// Mitsubishi GX Works2 project: plc_group6   PLC: FX3G

// global labels: Global1
VAR_GLOBAL
  switch10 AT X010 : BOOL;
  machineA AT M0 : BOOL;
  close_sys AT X005 : BOOL;
  sen_1 AT X001 : BOOL;
  sen_30 AT X002 : BOOL;
  sen_15 AT X003 : BOOL;
  sen_2 AT X004 : BOOL;
  zeluf_on AT Y004 : BOOL;
END_VAR
VAR_GLOBAL CONSTANT
  cream : INT := 700;
  chocolate : INT := 500;
  biscuit : INT := 100;
  ZeroConst : REAL;
END_VAR
VAR_GLOBAL
  TS1 : BOOL;
  TC1 AT TC1 : BOOL;
END_VAR
VAR_GLOBAL CONSTANT
  sec : INT := 40;
  sec_4 : INT := 40;
END_VAR
VAR_GLOBAL
  coil_y0 AT Y000 : BOOL;
  blink1 AT TS1 : BOOL;
  blink AT TC1 : BOOL;
  blink2 AT TC2 : BOOL;
  blink3 AT TS2 : BOOL;
  coil_y1 AT Y001 : BOOL;
  D_cream AT D1100 : REAL;
  D_chocolate AT D1102 : REAL;
  D_biscuit AT D1104 : REAL;
  end_day AT M1 : BOOL;
  start_day_button AT X007 : BOOL;
  start AT M2 : BOOL;
  start_day_lamp AT Y007 : BOOL;
  timer_tc3 AT TC3 : BOOL;
END_VAR
VAR_GLOBAL CONSTANT
  const_30_sec : INT := 30;
END_VAR
VAR_GLOBAL
  timer_ts3 AT TS3 : BOOL;
  blink_end AT M3 : BOOL;
END_VAR
VAR_GLOBAL CONSTANT
  cream_300 : REAL := 300;
  chocolate_240 : REAL := 240;
  biscuit_6 : REAL := 6;
END_VAR
VAR_GLOBAL
  D_ziluf AT D1106 : REAL;
  ziluf_button_x11 AT X011 : BOOL;
  ziluf_finish AT M4 : BOOL;
  D_tvila AT D1108 : REAL;
  sample_batton_x6 AT X006 : BOOL;
END_VAR
VAR_GLOBAL CONSTANT
  cream_700 : REAL := 700;
  chocolate_500 : REAL := 500;
  biscuit_100 : REAL := 100;
  nomalization : REAL := 400;
  nomalization_400 : REAL := 400;
END_VAR
VAR_GLOBAL
  sample_finish AT M5 : BOOL;
  finish_tvila_lamp AT Y003 : BOOL;
END_VAR
VAR_GLOBAL CONSTANT
  Double_tvila : REAL := 5;
  Double_amount : REAL := 240;
  normal_amount : REAL := 120;
END_VAR
VAR_GLOBAL
  timer_tc4 AT TC4 : BOOL;
END_VAR
VAR_GLOBAL CONSTANT
  sec_5 : INT := 50;
END_VAR
VAR_GLOBAL
  time_ts4 AT TS4 : BOOL;
  analog_input_1 AT D8280 : INT;
  blink_m5 AT M5 : BOOL;
  blink_m6 AT M6 : BOOL;
  data_analog_input_1 AT D1112 : INT;
  finish_tvila AT M7 : BOOL;
  start_ariza AT X000 : BOOL;
  counter_ariza_krembo AT CC0 : BOOL;
END_VAR
VAR_GLOBAL CONSTANT
  krembo_ariza_5 : INT := 5;
END_VAR
VAR_GLOBAL
  counter_ariza_krembo_5 AT CS0 : BOOL;
  counter_ariza_krembo_5_lamp AT Y002 : BOOL;
  counter_ariza_stop AT M8 : BOOL;
  krembo_sum AT D1114 : REAL;
END_VAR
VAR_GLOBAL CONSTANT
  add_krembo : REAL := 1;
END_VAR
VAR_GLOBAL
  counter_ariza_krembo_6 AT CC1 : BOOL;
END_VAR
VAR_GLOBAL CONSTANT
  krembo_ariza_6 : INT := 6;
END_VAR
VAR_GLOBAL
  check_stock AT M12 : BOOL;
END_VAR
VAR_GLOBAL CONSTANT
  multiply : INT := 40;
END_VAR
VAR_GLOBAL
  analog_output AT D8282 : INT;
  cream_input AT D1116 : REAL;
  chocolate_input AT D1118 : REAL;
  biscuit_input AT D1120 : REAL;
END_VAR
VAR_GLOBAL CONSTANT
  blink5 : INT := 5;
END_VAR
VAR_GLOBAL
  timer_tc5 AT TC5 : BOOL;
  help_blink1 AT M9 : BOOL;
  help_blink2 AT M10 : BOOL;
  help_blink3 AT M11 : BOOL;
  blink_tc6 AT TC6 : BOOL;
  blink_ts6 AT TS6 : BOOL;
  blink_tc7 AT TC7 : BOOL;
  blink_ts7 AT TS7 : BOOL;
  counter_ariza_krembo_6_stop AT CS1 : BOOL;
  sample AT D1121 : REAL;
END_VAR

// task Task_01 (event TRUE, interval 0, priority 31): POU_01

PROGRAM POU_01
VAR CONSTANT
  timer_ts4 : BOOL;
END_VAR
(* structured ladder/FBD written out as ST: instructions are called as NAME(EN, inputs, outputs); _pN, _eN, _tN stand for wires *)
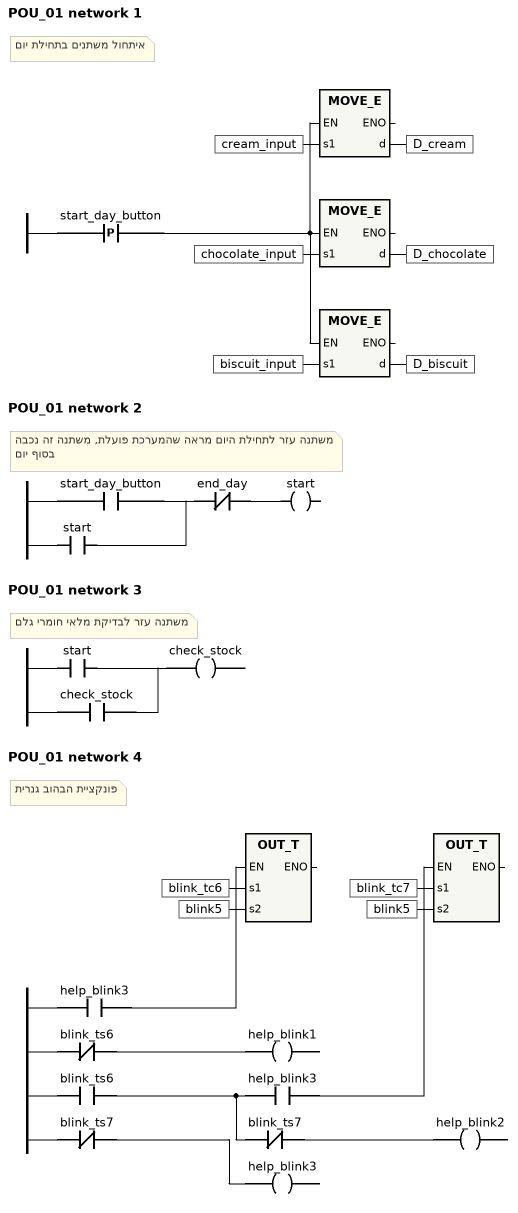
(* network 1 *)
(* איתחול משתנים בתחילת יום *)
_p1 := LDP(TRUE, start_day_button);
MOVE_E(_p1, cream_input, D_cream);
MOVE_E(_p1, chocolate_input, D_chocolate);
MOVE_E(_p1, biscuit_input, D_biscuit);
(* network 2 *)
(* משתנה עזר לתחילת היום מראה שהמערכת פועלת, משתנה זה נכבה בסוף יום *)
start := (start_day_button OR start) AND NOT end_day;
(* network 3 *)
(* משתנה עזר לבדיקת מלאי חומרי גלם *)
check_stock := start OR check_stock;
(* network 4 *)
(* פונקציית הבהוב גנרית *)
OUT_T(help_blink3, blink_tc6, blink5);
help_blink1 := NOT blink_ts6;
OUT_T(blink_ts6 AND help_blink3, blink_tc7, blink5);
help_blink2 := blink_ts6 AND NOT blink_ts7;
help_blink3 := NOT blink_ts7;
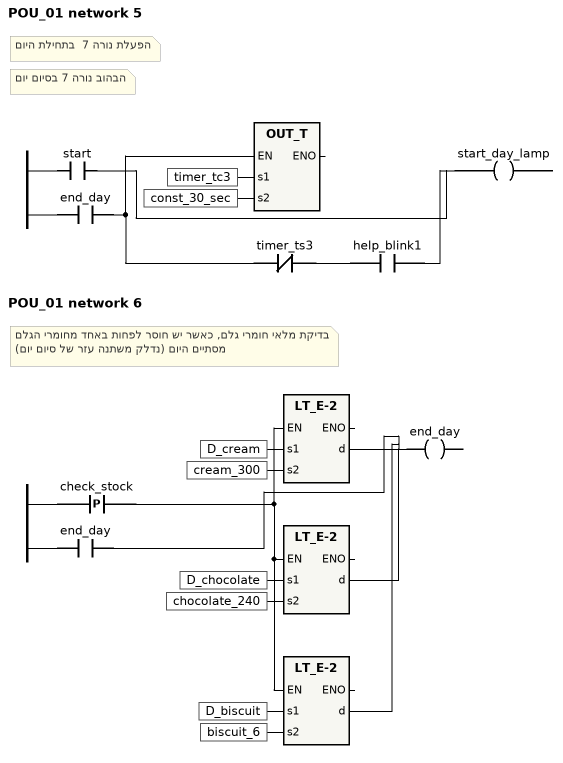
(* network 5 *)
(* הפעלת נורה 7  בתחילת היום *)
(* הבהוב נורה 7 בסיום יום *)
start_day_lamp := start OR (end_day AND NOT timer_ts3 AND help_blink1);
OUT_T(end_day, timer_tc3, const_30_sec);
(* network 6 *)
(* בדיקת מלאי חומרי גלם, כאשר יש חוסר לפחות באחד מחומרי הגלם  מסתיים היום (נדלק משתנה עזר של סיום יום) *)
_p1 := LDP(TRUE, check_stock);
LT_E(_p1, D_cream, cream_300, _t2);
LT_E(_p1, D_chocolate, chocolate_240, _t3);
LT_E(_p1, D_biscuit, biscuit_6, _t4);
end_day := _t2 OR _t3 OR _t4 OR end_day;
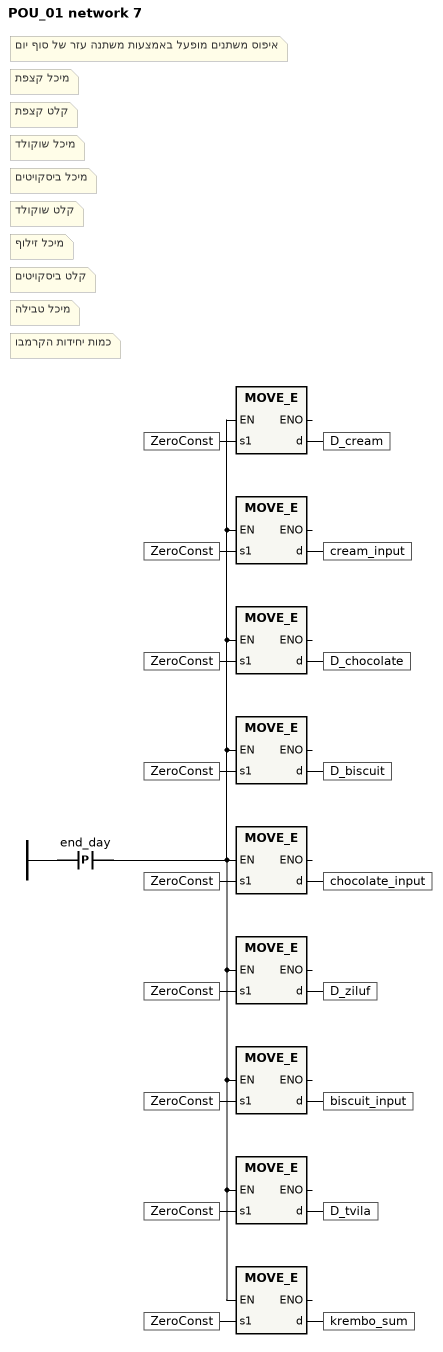
(* network 7 *)
(* איפוס משתנים מופעל באמצעות משתנה עזר של סוף יום *)
(* מיכל קצפת *)
(* קלט קצפת *)
(* מיכל שוקולד *)
(* מיכל ביסקויטים *)
(* קלט שוקולד *)
(* מיכל זילוף *)
(* קלט ביסקויטים *)
(* מיכל טבילה *)
(* כמות יחידות הקרמבו *)
_p1 := LDP(TRUE, end_day);
MOVE_E(_p1, ZeroConst, D_cream);
MOVE_E(_p1, ZeroConst, cream_input);
MOVE_E(_p1, ZeroConst, D_chocolate);
MOVE_E(_p1, ZeroConst, D_biscuit);
MOVE_E(_p1, ZeroConst, chocolate_input);
MOVE_E(_p1, ZeroConst, D_ziluf);
MOVE_E(_p1, ZeroConst, biscuit_input);
MOVE_E(_p1, ZeroConst, D_tvila);
MOVE_E(_p1, ZeroConst, krembo_sum);
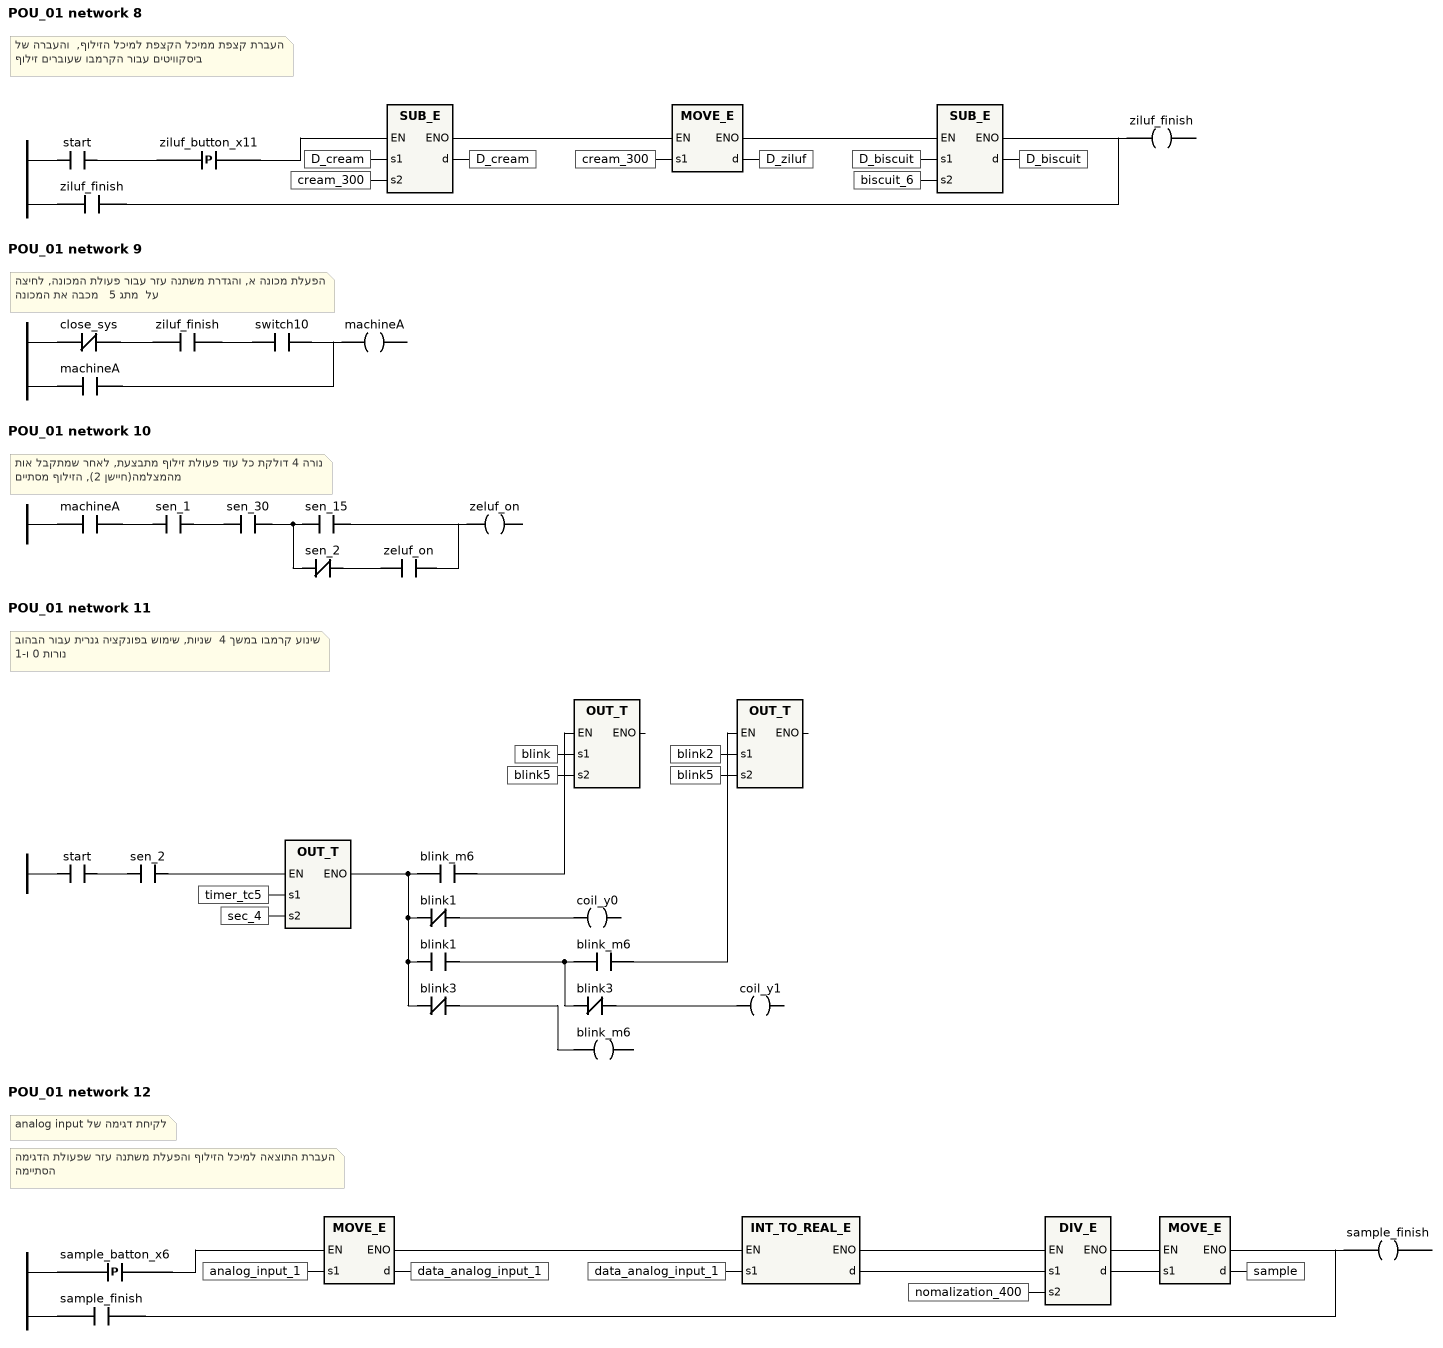
(* network 8 *)
(* העברת קצפת ממיכל הקצפת למיכל הזילוף,  והעברה של ביסקוויטים עבור הקרמבו שעוברים זילוף *)
_e1 := SUB_E(start AND LDP(TRUE, ziluf_button_x11), D_cream, cream_300, D_cream);
_e2 := MOVE_E(_e1, cream_300, D_ziluf);
_e3 := SUB_E(_e2, D_biscuit, biscuit_6, D_biscuit);
ziluf_finish := _e3 OR ziluf_finish;
(* network 9 *)
(* הפעלת מכונה א, והגדרת משתנה עזר עבור פעולת המכונה, לחיצה על  מתג 5   מכבה את המכונה *)
machineA := (NOT close_sys AND ziluf_finish AND switch10) OR machineA;
(* network 10 *)
(* נורה 4 דולקת כל עוד פעולת זילוף מתבצעת, לאחר שמתקבל אות מהמצלמה(חיישן 2), הזילוף מסתיים *)
_p1 := machineA AND sen_1 AND sen_30;
zeluf_on := (_p1 AND sen_15) OR (_p1 AND NOT sen_2 AND zeluf_on);
(* network 11 *)
(* שינוע קרמבו במשך 4  שניות, שימוש בפונקציה גנרית עבור הבהוב נורות 0 ו-1 *)
_e1 := OUT_T(start AND sen_2, timer_tc5, sec_4);
OUT_T(_e1 AND blink_m6, blink, blink5);
coil_y0 := _e1 AND NOT blink1;
_p2 := _e1 AND blink1;
OUT_T(_p2 AND blink_m6, blink2, blink5);
coil_y1 := _p2 AND NOT blink3;
blink_m6 := _e1 AND NOT blink3;
(* network 12 *)
(* לקיחת דגימה של analog input *)
(* העברת התוצאה למיכל הזילוף והפעלת משתנה עזר שפעולת הדגימה הסתיימה *)
_e1 := MOVE_E(LDP(TRUE, sample_batton_x6), analog_input_1, data_analog_input_1);
_e3 := INT_TO_REAL_E(_e1, data_analog_input_1, _t2);
_e5 := DIV_E(_e3, _t2, nomalization_400, _t4);
_e6 := MOVE_E(_e5, _t4, sample);
sample_finish := _e6 OR sample_finish;
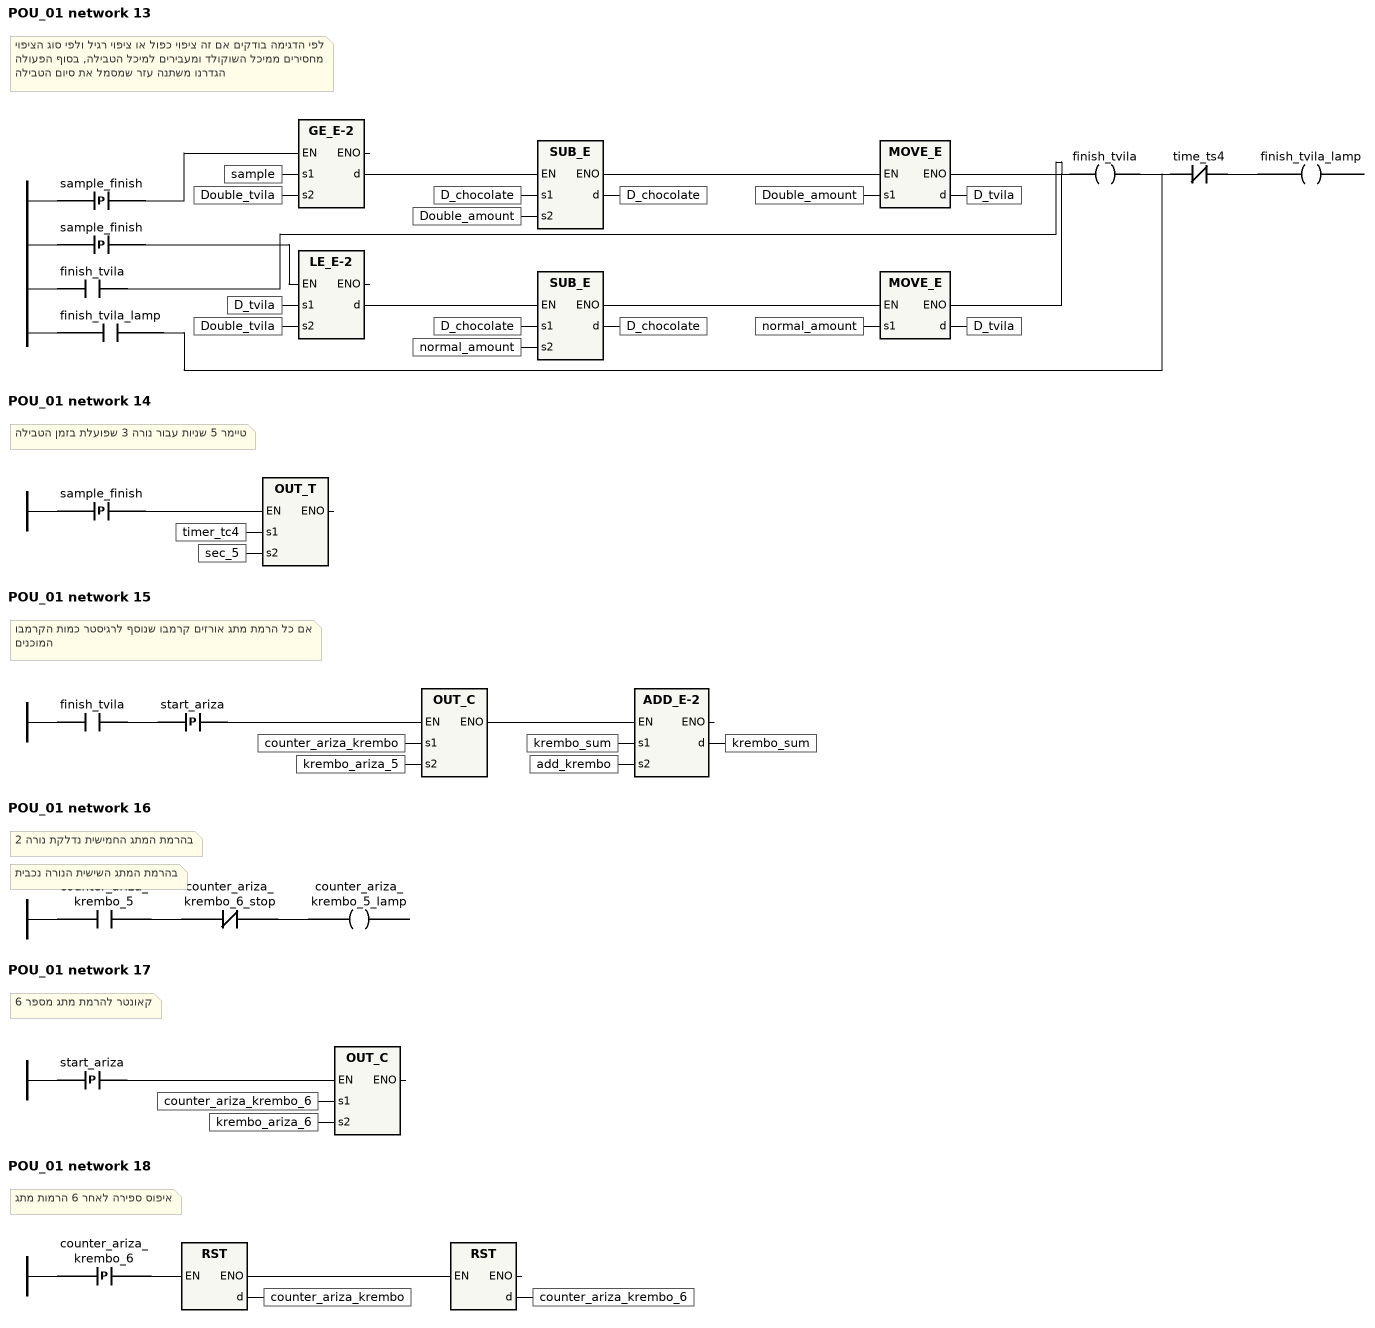
(* network 13 *)
(* לפי הדגימה בודקים אם זה ציפוי כפול או ציפוי רגיל ולפי סוג הציפוי מחסירים ממיכל השוקולד ומעבירים למיכל הטבילה, בסוף הפעולה  הגדרנו משתנה עזר שמסמל את סיום הטבילה *)
GE_E(LDP(TRUE, sample_finish), sample, Double_tvila, _t1);
_e2 := SUB_E(_t1, D_chocolate, Double_amount, D_chocolate);
_e3 := MOVE_E(_e2, Double_amount, D_tvila);
LE_E(LDP(TRUE, sample_finish), D_tvila, Double_tvila, _t4);
_e5 := SUB_E(_t4, D_chocolate, normal_amount, D_chocolate);
_e6 := MOVE_E(_e5, normal_amount, D_tvila);
_p7 := _e3 OR _e6 OR finish_tvila;
finish_tvila := _p7;
finish_tvila_lamp := (_p7 OR finish_tvila_lamp) AND NOT time_ts4;
(* network 14 *)
(* טיימר 5 שניות עבור נורה 3 שפועלת בזמן הטבילה *)
OUT_T(LDP(TRUE, sample_finish), timer_tc4, sec_5);
(* network 15 *)
(* אם כל הרמת מתג אורזים קרמבו שנוסף לרגיסטר כמות הקרמבו המוכנים *)
_e1 := OUT_C(finish_tvila AND LDP(TRUE, start_ariza), counter_ariza_krembo, krembo_ariza_5);
ADD_E(_e1, krembo_sum, add_krembo, krembo_sum);
(* network 16 *)
(* בהרמת המתג החמישית נדלקת נורה 2 *)
(* בהרמת המתג השישית הנורה נכבית *)
counter_ariza_krembo_5_lamp := counter_ariza_krembo_5 AND NOT counter_ariza_krembo_6_stop;
(* network 17 *)
(* קאונטר להרמת מתג מספר 6 *)
OUT_C(LDP(TRUE, start_ariza), counter_ariza_krembo_6, krembo_ariza_6);
(* network 18 *)
(* איפוס ספירה לאחר 6 הרמות מתג *)
_e1 := RST(LDP(TRUE, counter_ariza_krembo_6), counter_ariza_krembo);
RST(_e1, counter_ariza_krembo_6);
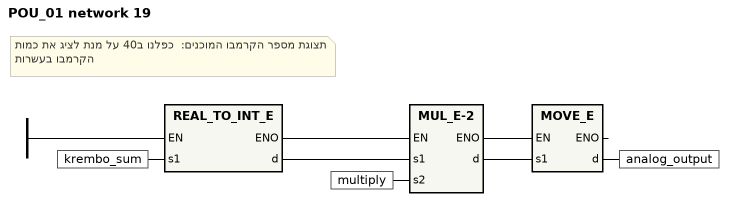
(* network 19 *)
(* תצוגת מספר הקרמבו המוכנים:  כפלנו ב40 על מנת לציג את כמות הקרמבו בעשרות *)
_e2 := REAL_TO_INT_E(TRUE, krembo_sum, _t1);
_e4 := MUL_E(_e2, _t1, multiply, _t3);
MOVE_E(_e4, _t3, analog_output);
END_PROGRAM
